// TIA Portal V16 export
// export: Created 2023-01-03T15:35:06.4312414Z, ExportSetting WithDefaults, DisplayName Totally Integrated Automation Portal, DisplayVersion V16, DisplayName TIA Portal Version Control Interface, DisplayVersion V16, DisplayName TIA Portal Openness, DisplayVersion V16, DisplayName STEP 7 Professional, DisplayVersion V16, DisplayName STEP 7 Safety, DisplayVersion V16, DisplayName WinCC Advanced, DisplayVersion V16
FUNCTION "MOTOR_MANUAL" : Void   // FC1, LAD
{ S7_Optimized_Access := 'TRUE' }
VERSION : 0.1
// stored: AutoNumber true, IsIECCheckEnabled false, SetENOAutomatically false, UDAEnableTagReadback false
   VAR_INPUT
      "PLANT ON" : Bool;
      "NO EMERGENCY" : Bool;
      "MANUAL MODE" : Bool;
      "CYLINDER M4 RESTRACTED" : Bool;
      "FORWARD PB" : Bool;
      "REVERSED PB" : Bool;
   END_VAR
   VAR_OUTPUT
      FORWARD : Bool;
      REVERSED : Bool;
   END_VAR
BEGIN

REGION Network 1: MOTOR DRIVE IN FORWARD DIRECTION
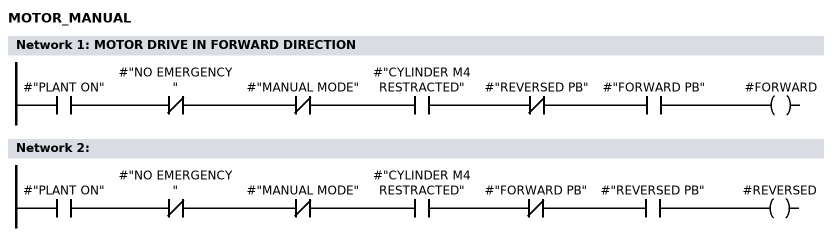
   RUNG wire#powerrail
      Contact( #"PLANT ON" )
      I_Contact( #"NO EMERGENCY" )
      I_Contact( #"MANUAL MODE" )
      Contact( #"CYLINDER M4 RESTRACTED" )
      I_Contact( #"REVERSED PB" )
      Contact( #"FORWARD PB" )
      Coil( #FORWARD )
   END_RUNG
   // the same network as SCL:
   #FORWARD := #"PLANT ON" AND NOT #"NO EMERGENCY" AND NOT #"MANUAL MODE" AND #"CYLINDER M4 RESTRACTED" AND NOT #"REVERSED PB" AND #"FORWARD PB";
END_REGION

REGION Network 2
   RUNG wire#powerrail
      Contact( #"PLANT ON" )
      I_Contact( #"NO EMERGENCY" )
      I_Contact( #"MANUAL MODE" )
      Contact( #"CYLINDER M4 RESTRACTED" )
      I_Contact( #"FORWARD PB" )
      Contact( #"REVERSED PB" )
      Coil( #REVERSED )
   END_RUNG
   // the same network as SCL:
   #REVERSED := #"PLANT ON" AND NOT #"NO EMERGENCY" AND NOT #"MANUAL MODE" AND #"CYLINDER M4 RESTRACTED" AND NOT #"FORWARD PB" AND #"REVERSED PB";
END_REGION
END_FUNCTION
